FUNCTION_BLOCK fbPressing
VAR_INPUT
	SafetyOk			: BOOL;
	ResetCmd			: BOOL;
	AutoCycle			: BOOL;
	ManualCmd			: BOOL;
END_VAR
VAR_OUTPUT
	ResetCompleted 		: BOOL;
		
END_VAR
VAR
	
	ForceReached			AT %I* :BOOL;
	
	AdvancePress			AT %Q* :BOOL;
	
	State					: INT := 0;

END_VAR

END_FUNCTION_BLOCK

(* stored: Version 1.1.0.1, ProductVersion 3.1.4022.18
   POU fbPressing: Id {bc34757d-9fed-470c-8097-6f136cd894a9}, SpecialFunc None *)
